PROGRAM MAIN
VAR
	Counter: INT;
	
	Safety_Reset AT %Q*:BOOL;
	Safety_Run AT %Q*:BOOL :=TRUE;
	Safety_ErroAck AT %Q*:BOOL;
END_VAR

Counter:=Counter+1;


//Safety_BckpRstr();

END_PROGRAM

(* stored: Version 1.1.0.1, ProductVersion 3.1.4024.12
   POU MAIN: Id {a006fe57-da36-4aba-b269-66eb17a3ab15}, SpecialFunc None *)
